FUNCTION_BLOCK PID_LEVEL (* Basic FB with empty ECC *)
  (* Standard: 61499-2 *)
  (* Version 1.0, 2026-03-26, guilh *)
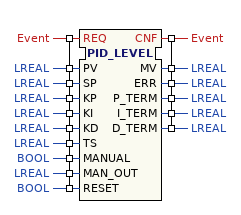
  EVENT_INPUT
    REQ WITH PV, SP, KP, KI, KD, TS, MANUAL, MAN_OUT, RESET; (* When receives REQ calculates PID *)
  END_EVENT
  EVENT_OUTPUT
    CNF WITH MV, ERR, P_TERM, I_TERM, D_TERM; (* When finish calculation it sends *)
  END_EVENT
  VAR_INPUT
    PV : LREAL; (* Process variable, measure level *)
    SP : LREAL; (* Setpoint *)
    KP : LREAL;
    KI : LREAL;
    KD : LREAL;
    TS : LREAL; (* Period defined in seconds *)
    MANUAL : BOOL;
    MAN_OUT : LREAL;
    RESET : BOOL;
  END_VAR
  VAR_OUTPUT
    MV : LREAL; (* PID output from 0 to 100 *)
    ERR : LREAL;
    P_TERM : LREAL;
    I_TERM : LREAL;
    D_TERM : LREAL;
  END_VAR
  VAR
    e_prev : LREAL := 0.0; (* guarda o erro anterior para calcular a derivada *)
    i_acc : LREAL := 0.0; (* guarda a integral acumulada *)
    u_raw : LREAL := 0.0; (* guarda a saída antes da saturação *)
  END_VAR
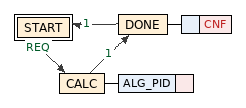
  EC_STATES
    START; (* Initial State *)
    CALC : ALG_PID;
    DONE : -> CNF;
  END_STATES
  EC_TRANSITIONS
    START TO CALC := REQ;
    CALC TO DONE := 1;
    DONE TO START := 1;
  END_TRANSITIONS
  ALGORITHM ALG_PID IN ST:
IF RESET THEN
    i_acc := 0.0;
    e_prev := 0.0;
END_IF;

IF MANUAL THEN
    MV := MAN_OUT;

    IF MV > 100.0 THEN
        MV := 100.0;
    ELSIF MV < 0.0 THEN
        MV := 0.0;
    END_IF;

    ERR := SP - PV;
    P_TERM := 0.0;
    I_TERM := 0.0;
    D_TERM := 0.0;

ELSE
    ERR := SP - PV;

    P_TERM := KP * ERR;

    i_acc := i_acc + (ERR * TS);
    I_TERM := KI * i_acc;

    D_TERM := KD * ((ERR - e_prev) / TS);

    u_raw := P_TERM + I_TERM + D_TERM;

    IF u_raw > 100.0 THEN
        MV := 100.0;
    ELSIF u_raw < 0.0 THEN
        MV := 0.0;
    ELSE
        MV := u_raw;
    END_IF;

    e_prev := ERR;
END_IF;
  END_ALGORITHM
END_FUNCTION_BLOCK
